(* Logix 5000 project; controller PROJECT2 Emulate 5570 rev 30.12; software revision 30.01; part 2 of 3 *)

ADD_ON_INSTRUCTION AOI_SIMAnalogSensor_OnOff   (* revision 1.0 *)
VAR_IN_OUT
   Sensor : REAL; {required}
END_VAR
VAR_INPUT
   RampUpTime : DINT; {required}
   RampDwnTime : DINT; {required}
   Min : REAL; {required}
   Max : REAL; {required}
   Target : REAL; {visible}
   Tolerance : REAL; {visible}
   Fluctuation : REAL; {access None, visible}
   Activate : BOOL; {access None}
END_VAR
VAR
   RampUpTimer : TIMER; {access None}
   RampDwnTimer : TIMER; {access None}
   FluctuateTimer : TIMER; {access None}
   FluctuateONS : BOOL; {access None}
   CurrentValue : REAL; {access Read Only}
   RampDwnTriggerONS : BOOL; {access Read Only}
   RampDwnTriggerPulse : BOOL; {access Read Only}
   RampUpTriggerONS : BOOL; {access Read Only}
   RampUpTriggerPulse : BOOL; {access Read Only}
   RandomNumber : DINT; {access Read Only}
   RandomTarget : REAL; {access Read Only}
   RandomIntermediate : DINT; {access Read Only}
   ScaledRampDwnTime : REAL; {access Read Only}
   ScaledRampUpTime : REAL; {access Read Only}
   Fluctuate : BOOL; {access None}
   LowerTargetTriggerONS : BOOL; {access None}
   OldTarget : REAL; {access None}
   RaiseTargetTriggerONS : BOOL; {access None}
END_VAR

ROUTINE Logic   (* ladder *)
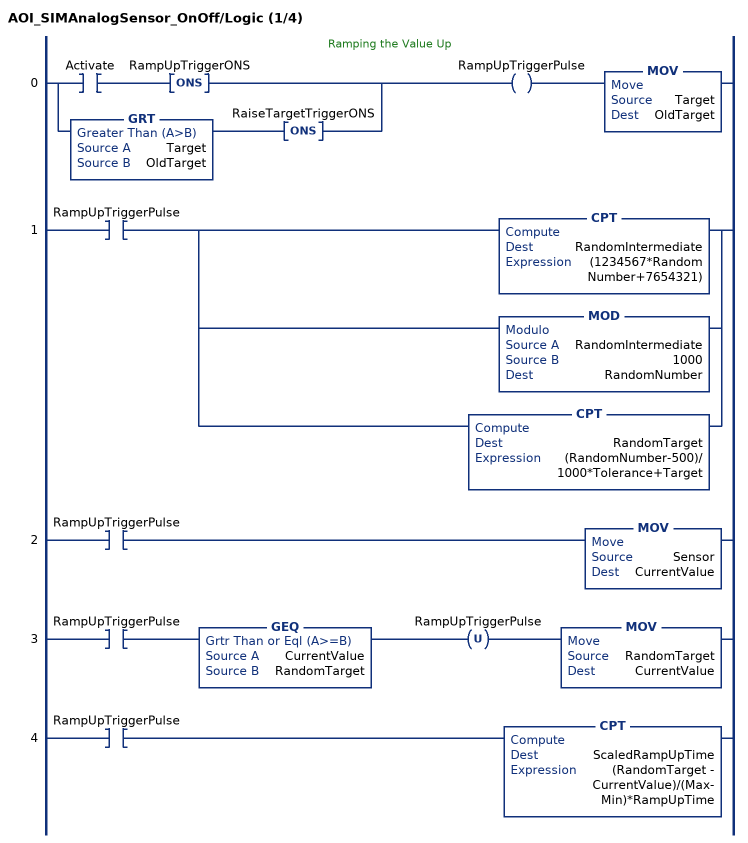
   // Ramping the Value Up
   0: [XIC(Activate) ONS(RampUpTriggerONS) ,GRT(Target,OldTarget) ONS(RaiseTargetTriggerONS) ]OTE(RampUpTriggerPulse)MOV(Target,OldTarget);
   1: XIC(RampUpTriggerPulse)[CPT(RandomIntermediate,(1234567*RandomNumber+7654321)) ,MOD(RandomIntermediate,1000,RandomNumber) ,CPT(RandomTarget,(RandomNumber-500)/1000*Tolerance+Target) ];
   2: XIC(RampUpTriggerPulse)MOV(Sensor,CurrentValue);
   3: XIC(RampUpTriggerPulse)GEQ(CurrentValue,RandomTarget)OTU(RampUpTriggerPulse)MOV(RandomTarget,CurrentValue);
   4: XIC(RampUpTriggerPulse)CPT(ScaledRampUpTime,(RandomTarget - CurrentValue)/(Max-Min)*RampUpTime);
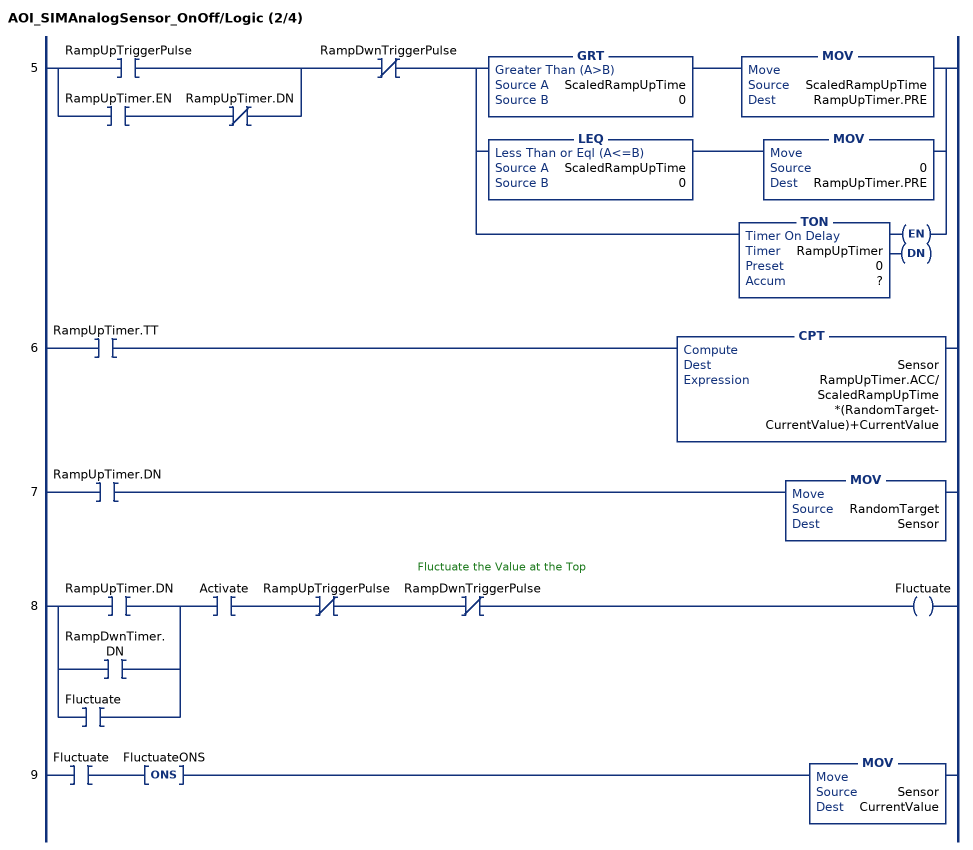
   5: [XIC(RampUpTriggerPulse) ,XIC(RampUpTimer.EN) XIO(RampUpTimer.DN) ]XIO(RampDwnTriggerPulse)[GRT(ScaledRampUpTime,0) MOV(ScaledRampUpTime,RampUpTimer.PRE) ,LEQ(ScaledRampUpTime,0) MOV(0,RampUpTimer.PRE) ,TON(RampUpTimer,?,?) ];
   6: XIC(RampUpTimer.TT)CPT(Sensor,RampUpTimer.ACC/ScaledRampUpTime *(RandomTarget-CurrentValue)+CurrentValue);
   7: XIC(RampUpTimer.DN)MOV(RandomTarget,Sensor);
   // Fluctuate the Value at the Top
   8: [XIC(RampUpTimer.DN) ,XIC(RampDwnTimer.DN) ,XIC(Fluctuate) ]XIC(Activate)XIO(RampUpTriggerPulse)XIO(RampDwnTriggerPulse)OTE(Fluctuate);
   9: XIC(Fluctuate)ONS(FluctuateONS)MOV(Sensor,CurrentValue);
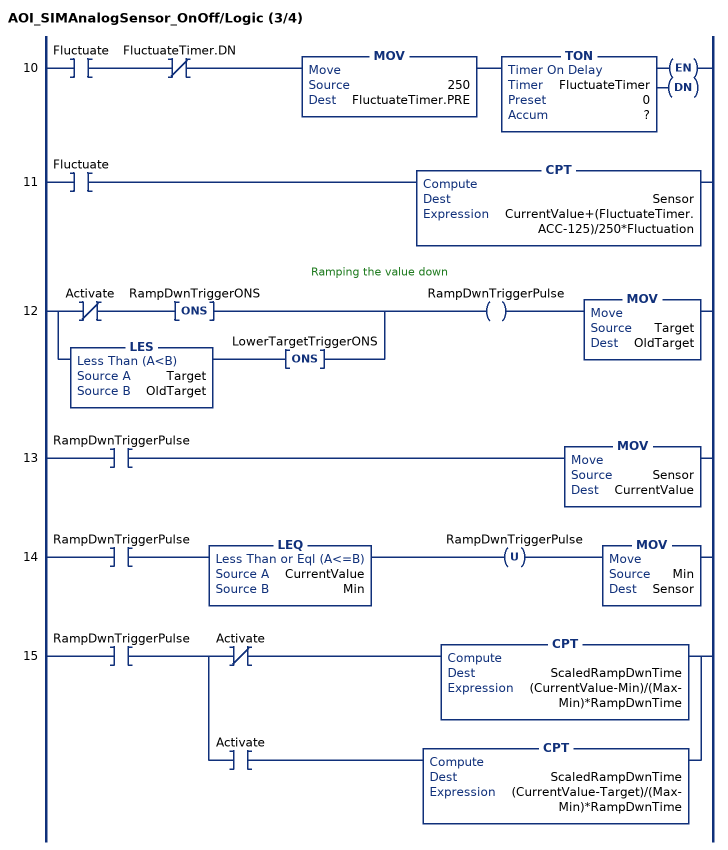
   10: XIC(Fluctuate)XIO(FluctuateTimer.DN)MOV(250,FluctuateTimer.PRE)TON(FluctuateTimer,?,?);
   11: XIC(Fluctuate)CPT(Sensor,CurrentValue+(FluctuateTimer.ACC-125)/250*Fluctuation);
   // Ramping the value down
   12: [XIO(Activate) ONS(RampDwnTriggerONS) ,LES(Target,OldTarget) ONS(LowerTargetTriggerONS) ]OTE(RampDwnTriggerPulse)MOV(Target,OldTarget);
   13: XIC(RampDwnTriggerPulse)MOV(Sensor,CurrentValue);
   14: XIC(RampDwnTriggerPulse)LEQ(CurrentValue,Min)OTU(RampDwnTriggerPulse)MOV(Min,Sensor);
   15: XIC(RampDwnTriggerPulse)[XIO(Activate) CPT(ScaledRampDwnTime,(CurrentValue-Min)/(Max-Min)*RampDwnTime) ,XIC(Activate) CPT(ScaledRampDwnTime,(CurrentValue-Target)/(Max-Min)*RampDwnTime) ];
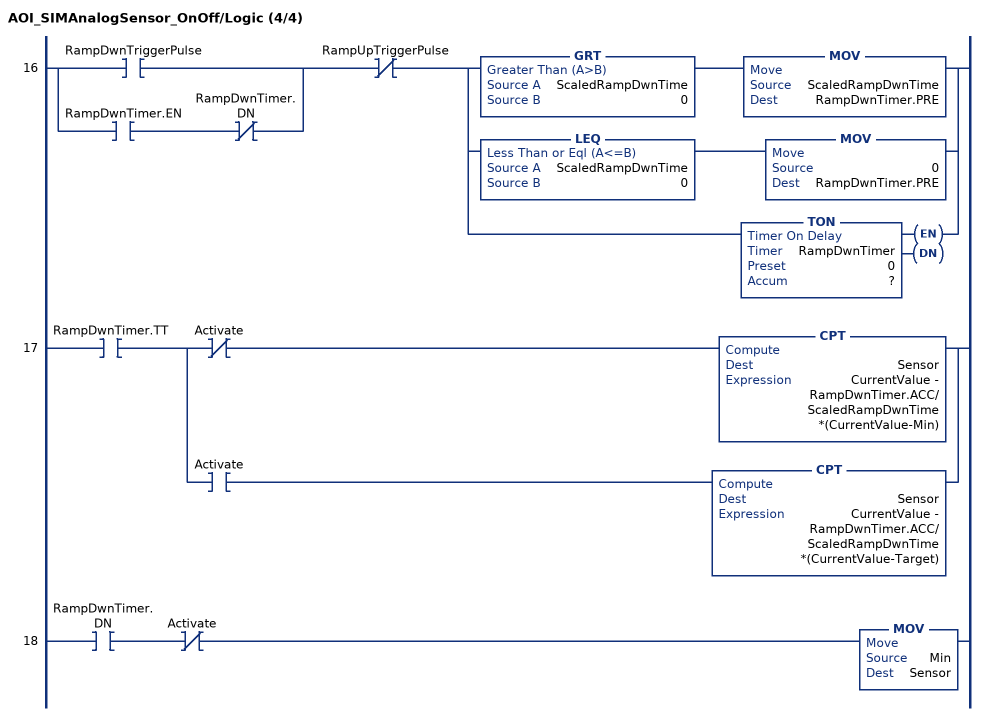
   16: [XIC(RampDwnTriggerPulse) ,XIC(RampDwnTimer.EN) XIO(RampDwnTimer.DN) ]XIO(RampUpTriggerPulse)[GRT(ScaledRampDwnTime,0) MOV(ScaledRampDwnTime,RampDwnTimer.PRE) ,LEQ(ScaledRampDwnTime,0) MOV(0,RampDwnTimer.PRE) ,TON(RampDwnTimer,?,?) ];
   17: XIC(RampDwnTimer.TT)[XIO(Activate) CPT(Sensor,CurrentValue - RampDwnTimer.ACC/ScaledRampDwnTime *(CurrentValue-Min)) ,XIC(Activate) CPT(Sensor,CurrentValue - RampDwnTimer.ACC/ScaledRampDwnTime *(CurrentValue-Target)) ];
   18: XIC(RampDwnTimer.DN)XIO(Activate)MOV(Min,Sensor);
END_ROUTINE
END_ADD_ON_INSTRUCTION

ADD_ON_INSTRUCTION AOI_SIMAnalogSensor_Profile   (* revision 1.0 *)
VAR_IN_OUT
   Sensor : REAL; {required}
END_VAR
VAR_INPUT
   RampUpTime : DINT; {required}
   RampDwnTime : DINT; {required}
   Min : REAL; {required}
   Max : REAL; {required}
   Target : REAL; {visible}
   Tolerance : REAL; {visible}
   Fluctuation : REAL; {access None, visible}
   Activate : BOOL; {access None}
END_VAR
VAR
   RampUpTimer : TIMER; {access None}
   RampDwnTimer : TIMER; {access None}
   FluctuateTimer : TIMER; {access None}
   FluctuateONS : BOOL; {access None}
   CurrentValue : REAL; {access Read Only}
   RampDwnTriggerONS : BOOL; {access Read Only}
   RampDwnTriggerPulse : BOOL; {access Read Only}
   RampUpTriggerONS : BOOL; {access Read Only}
   RampTriggerPulse : BOOL; {access Read Only}
   RandomNumber : DINT; {access Read Only}
   RandomTarget : REAL; {access Read Only}
   RandomIntermediate : DINT; {access Read Only}
   ScaledRampDwnTime : REAL; {access Read Only}
   ScaledRampUpTime : REAL; {access Read Only}
   Fluctuate : BOOL; {access None}
   LowerTargetTriggerONS : BOOL; {access None}
   OldTarget : REAL; {access None}
   RaiseTargetTriggerONS : BOOL; {access None}
END_VAR

ROUTINE Logic   (* ladder *)
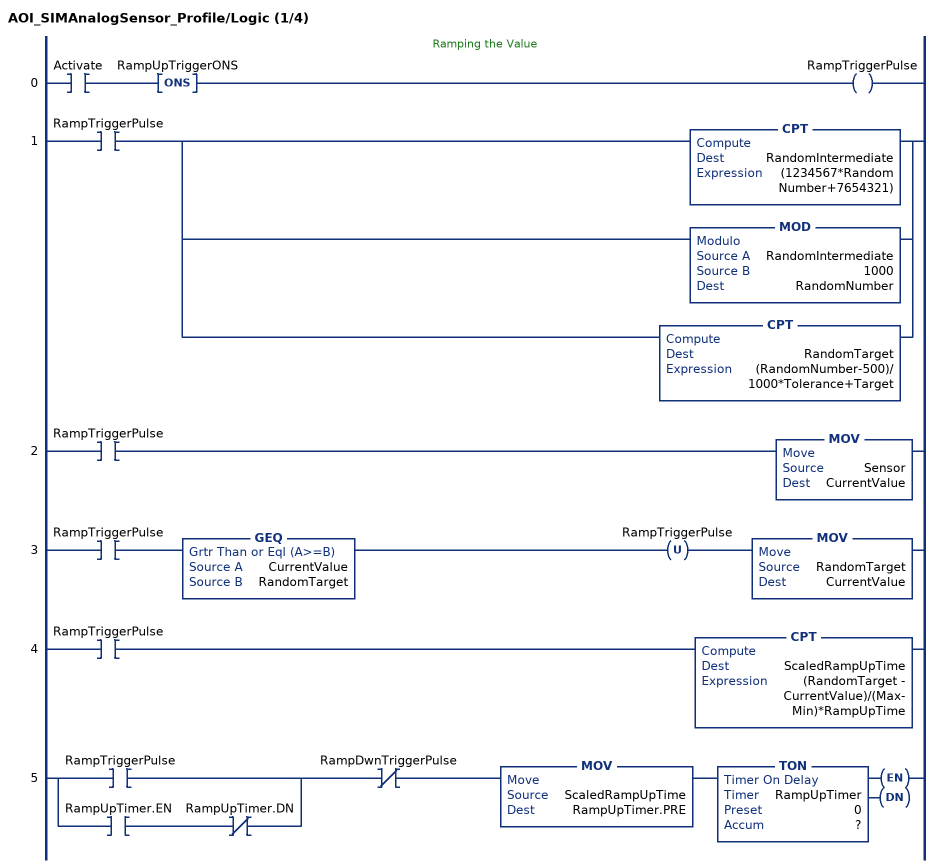
   // Ramping the Value
   0: XIC(Activate)ONS(RampUpTriggerONS)OTE(RampTriggerPulse);
   1: XIC(RampTriggerPulse)[CPT(RandomIntermediate,(1234567*RandomNumber+7654321)) ,MOD(RandomIntermediate,1000,RandomNumber) ,CPT(RandomTarget,(RandomNumber-500)/1000*Tolerance+Target) ];
   2: XIC(RampTriggerPulse)MOV(Sensor,CurrentValue);
   3: XIC(RampTriggerPulse)GEQ(CurrentValue,RandomTarget)OTU(RampTriggerPulse)MOV(RandomTarget,CurrentValue);
   4: XIC(RampTriggerPulse)CPT(ScaledRampUpTime,(RandomTarget - CurrentValue)/(Max-Min)*RampUpTime);
   5: [XIC(RampTriggerPulse) ,XIC(RampUpTimer.EN) XIO(RampUpTimer.DN) ]XIO(RampDwnTriggerPulse)MOV(ScaledRampUpTime,RampUpTimer.PRE)TON(RampUpTimer,?,?);
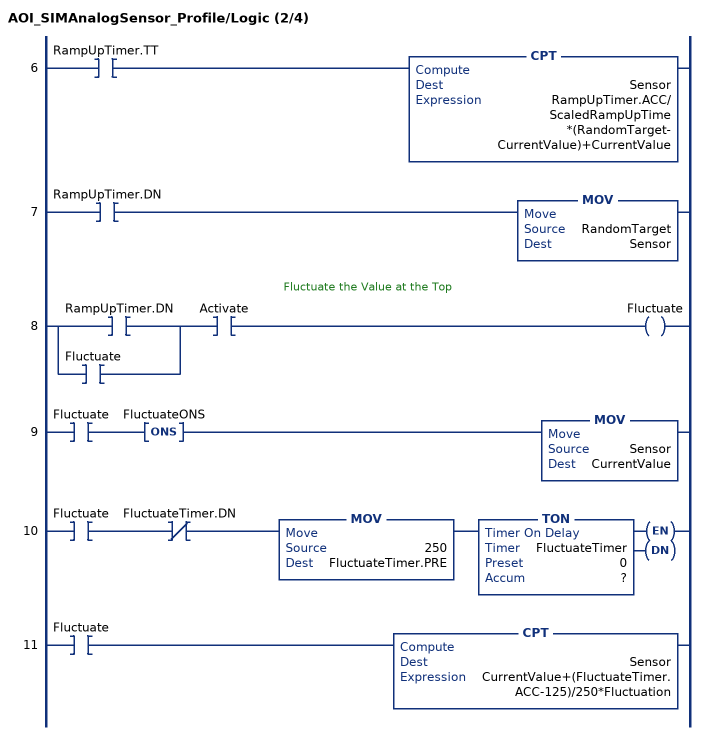
   6: XIC(RampUpTimer.TT)CPT(Sensor,RampUpTimer.ACC/ScaledRampUpTime *(RandomTarget-CurrentValue)+CurrentValue);
   7: XIC(RampUpTimer.DN)MOV(RandomTarget,Sensor);
   // Fluctuate the Value at the Top
   8: [XIC(RampUpTimer.DN) ,XIC(Fluctuate) ]XIC(Activate)OTE(Fluctuate);
   9: XIC(Fluctuate)ONS(FluctuateONS)MOV(Sensor,CurrentValue);
   10: XIC(Fluctuate)XIO(FluctuateTimer.DN)MOV(250,FluctuateTimer.PRE)TON(FluctuateTimer,?,?);
   11: XIC(Fluctuate)CPT(Sensor,CurrentValue+(FluctuateTimer.ACC-125)/250*Fluctuation);
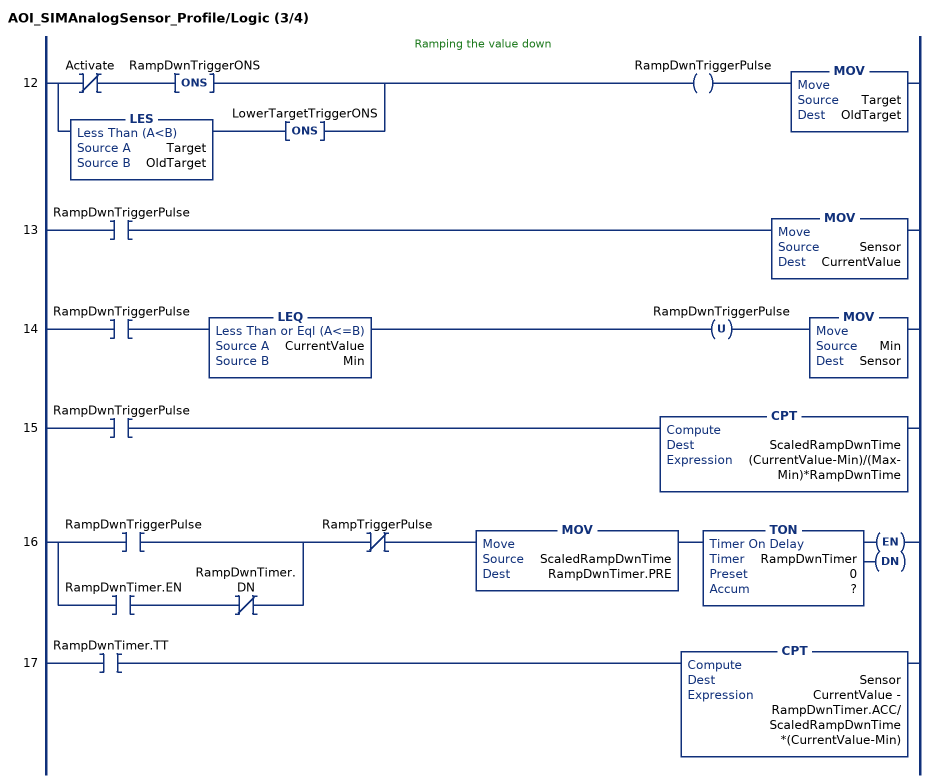
   // Ramping the value down
   12: [XIO(Activate) ONS(RampDwnTriggerONS) ,LES(Target,OldTarget) ONS(LowerTargetTriggerONS) ]OTE(RampDwnTriggerPulse)MOV(Target,OldTarget);
   13: XIC(RampDwnTriggerPulse)MOV(Sensor,CurrentValue);
   14: XIC(RampDwnTriggerPulse)LEQ(CurrentValue,Min)OTU(RampDwnTriggerPulse)MOV(Min,Sensor);
   15: XIC(RampDwnTriggerPulse)CPT(ScaledRampDwnTime,(CurrentValue-Min)/(Max-Min)*RampDwnTime);
   16: [XIC(RampDwnTriggerPulse) ,XIC(RampDwnTimer.EN) XIO(RampDwnTimer.DN) ]XIO(RampTriggerPulse)MOV(ScaledRampDwnTime,RampDwnTimer.PRE)TON(RampDwnTimer,?,?);
   17: XIC(RampDwnTimer.TT)CPT(Sensor,CurrentValue - RampDwnTimer.ACC/ScaledRampDwnTime *(CurrentValue-Min));
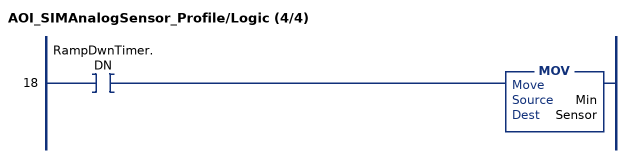
   18: XIC(RampDwnTimer.DN)MOV(Min,Sensor);
END_ROUTINE
END_ADD_ON_INSTRUCTION

ADD_ON_INSTRUCTION AOI_SIMPartSensor   (* revision 1.0 *)
VAR_OUTPUT
   Animation : DINT; {access Read Only, visible}
   Sensor : BOOL; {access Read Only, visible}
END_VAR
VAR_INPUT
   TP_ToggleSensorPB : BOOL;
   SensorON : BOOL;
   SensorOFF : BOOL;
   ONDelayTime : DINT; {visible}
   OFFDelayTime : DINT; {visible}
END_VAR
VAR_OUTPUT
   Sensor_Input : BOOL; {access Read Only, required}
END_VAR
VAR_INPUT
   SimEnabled : BOOL; {required}
   SensorONPause : BOOL;
   SensorOFFPause : BOOL;
END_VAR
VAR
   TmrON : TIMER; {access None}
   TmrOFF : TIMER; {access None}
   TP_AutoToggleSensorOFFPulse : BOOL; {access None}
   TP_AutoToggleSensorONPulse : BOOL; {access None}
   TP_AutoToggleSensorON_ONS : BOOL; {access None}
   TP_AutoToggleSensorOFF_ONS : BOOL; {access None}
   SensorOFF_ONS : BOOL; {access None}
   SensorON_ONS : BOOL; {access None}
   SensorWaitingToTurnON : BOOL; {access None}
   SensorWaitingToTurnOFF : BOOL; {access None}
   TP_ManualToggleSensorON_PULSE : BOOL; {access None}
   TP_ManualToggleSensor_ONS : BOOL; {access None}
   TP_ManualToggleSensorOFF_PULSE : BOOL; {access None}
   TP_ManualToggleSensorOFF_ONS : BOOL; {access None}
END_VAR

ROUTINE Logic   (* ladder *)
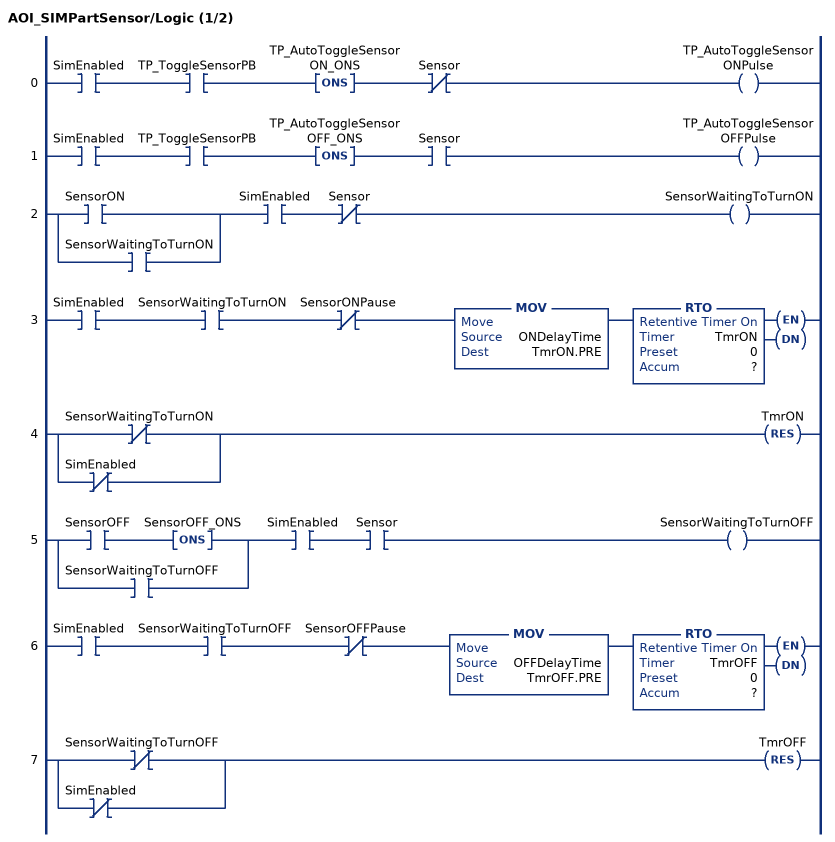
   0: XIC(SimEnabled)XIC(TP_ToggleSensorPB)ONS(TP_AutoToggleSensorON_ONS)XIO(Sensor)OTE(TP_AutoToggleSensorONPulse);
   1: XIC(SimEnabled)XIC(TP_ToggleSensorPB)ONS(TP_AutoToggleSensorOFF_ONS)XIC(Sensor)OTE(TP_AutoToggleSensorOFFPulse);
   2: [XIC(SensorON) ,XIC(SensorWaitingToTurnON) ]XIC(SimEnabled)XIO(Sensor)OTE(SensorWaitingToTurnON);
   3: XIC(SimEnabled)XIC(SensorWaitingToTurnON)XIO(SensorONPause)MOV(ONDelayTime,TmrON.PRE)RTO(TmrON,?,?);
   4: [XIO(SensorWaitingToTurnON) ,XIO(SimEnabled) ]RES(TmrON);
   5: [XIC(SensorOFF) ONS(SensorOFF_ONS) ,XIC(SensorWaitingToTurnOFF) ]XIC(SimEnabled)XIC(Sensor)OTE(SensorWaitingToTurnOFF);
   6: XIC(SimEnabled)XIC(SensorWaitingToTurnOFF)XIO(SensorOFFPause)MOV(OFFDelayTime,TmrOFF.PRE)RTO(TmrOFF,?,?);
   7: [XIO(SensorWaitingToTurnOFF) ,XIO(SimEnabled) ]RES(TmrOFF);
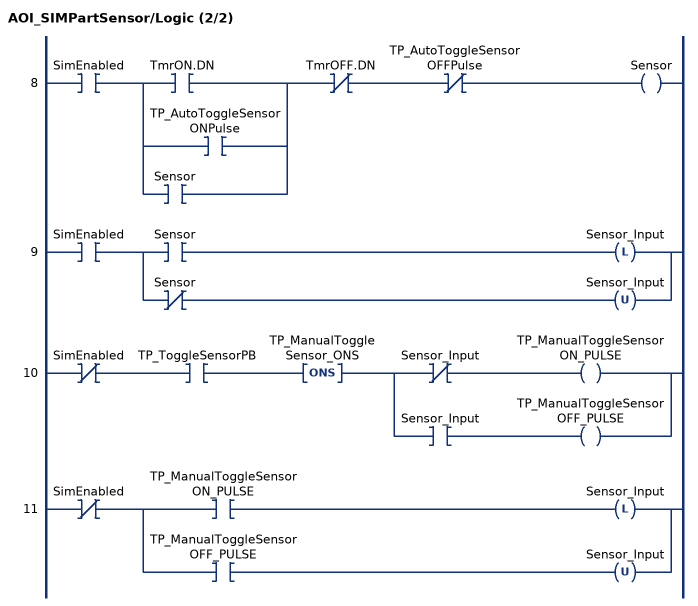
   8: XIC(SimEnabled)[XIC(TmrON.DN) ,XIC(TP_AutoToggleSensorONPulse) ,XIC(Sensor) ]XIO(TmrOFF.DN)XIO(TP_AutoToggleSensorOFFPulse)OTE(Sensor);
   9: XIC(SimEnabled)[XIC(Sensor) OTL(Sensor_Input) ,XIO(Sensor) OTU(Sensor_Input) ];
   10: XIO(SimEnabled)XIC(TP_ToggleSensorPB)ONS(TP_ManualToggleSensor_ONS)[XIO(Sensor_Input) OTE(TP_ManualToggleSensorON_PULSE) ,XIC(Sensor_Input) OTE(TP_ManualToggleSensorOFF_PULSE) ];
   11: XIO(SimEnabled)[XIC(TP_ManualToggleSensorON_PULSE) OTL(Sensor_Input) ,XIC(TP_ManualToggleSensorOFF_PULSE) OTU(Sensor_Input) ];
END_ROUTINE
END_ADD_ON_INSTRUCTION

ADD_ON_INSTRUCTION AOI_SIMPartTravel   (* revision 1.0 *)
VAR_OUTPUT
   Travelling : BOOL; {access Read Only, visible}
END_VAR
VAR_INPUT
   TravelTime : DINT; {required}
END_VAR
VAR_OUTPUT
   Animation : DINT; {access Read Only, visible}
END_VAR
VAR_INPUT
   TP_PB : BOOL;
   TravelON : BOOL;
   TravelOFF : BOOL;
   SimEnabled : BOOL; {required}
END_VAR
VAR_OUTPUT
   TravellingFirstHalf : BOOL; {access Read Only}
   TravellingLastHalf : BOOL; {access Read Only}
   TravellingLastQuarter : BOOL; {access Read Only}
   TravellingFirstQuarter : BOOL; {access Read Only}
   TravellingFirst10Percent : BOOL; {access Read Only}
   TravellingLast10Percent : BOOL; {access Read Only}
END_VAR
VAR_INPUT
   Pause : BOOL;
END_VAR
VAR_OUTPUT
   Done : BOOL; {access Read Only}
END_VAR
VAR
   Tmr : TIMER := (PRE := 1500); {access None}
   TravelON_ONS : BOOL; {access None}
   TravelTime75Percent : DINT; {access None}
   TravelTime50Percent : DINT; {access None}
   TravelTime25Percent : DINT; {access None}
   TravelTime10Percent : DINT; {access Read Only}
   TravelTime90Percent : DINT; {access Read Only}
   DonePulse : TIMER := (PRE := 250); {access None}
   TP_AutoToggleTravellingON_ONS : BOOL; {access None}
   TP_AutoToggleTravellingONPulse : BOOL; {access None}
   TP_AutoToggleTravellingOFFPulse : BOOL; {access None}
   TP_AutoToggleTravellingOFF_ONS : BOOL; {access None}
END_VAR

ROUTINE Logic   (* ladder *)
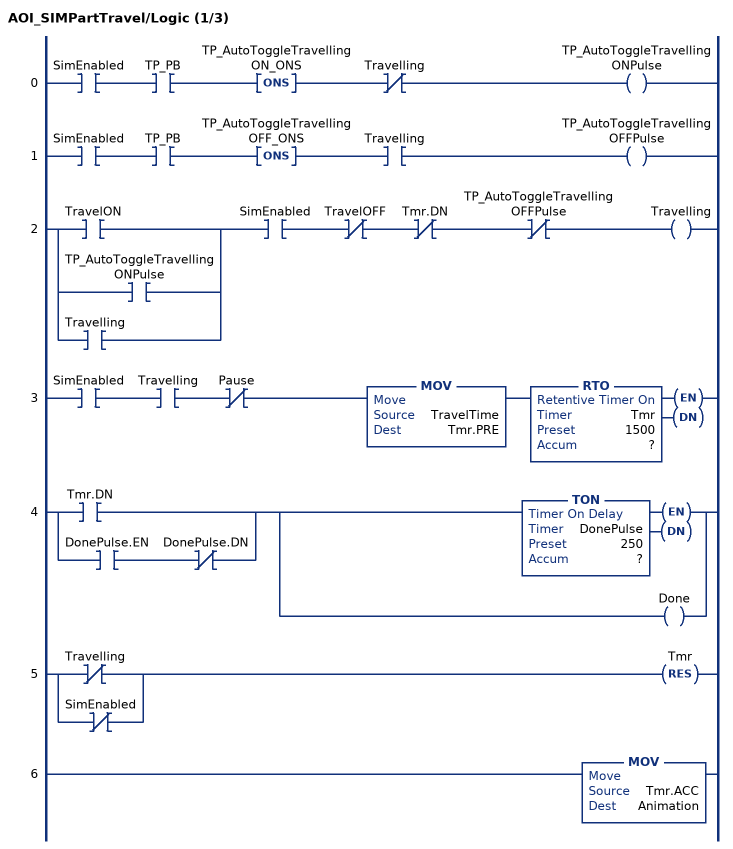
   0: XIC(SimEnabled)XIC(TP_PB)ONS(TP_AutoToggleTravellingON_ONS)XIO(Travelling)OTE(TP_AutoToggleTravellingONPulse);
   1: XIC(SimEnabled)XIC(TP_PB)ONS(TP_AutoToggleTravellingOFF_ONS)XIC(Travelling)OTE(TP_AutoToggleTravellingOFFPulse);
   2: [XIC(TravelON) ,XIC(TP_AutoToggleTravellingONPulse) ,XIC(Travelling) ]XIC(SimEnabled)XIO(TravelOFF)XIO(Tmr.DN)XIO(TP_AutoToggleTravellingOFFPulse)OTE(Travelling);
   3: XIC(SimEnabled)XIC(Travelling)XIO(Pause)MOV(TravelTime,Tmr.PRE)RTO(Tmr,?,?);
   4: [XIC(Tmr.DN) ,XIC(DonePulse.EN) XIO(DonePulse.DN) ][TON(DonePulse,?,?) ,OTE(Done) ];
   5: [XIO(Travelling) ,XIO(SimEnabled) ]RES(Tmr);
   6: MOV(Tmr.ACC,Animation);
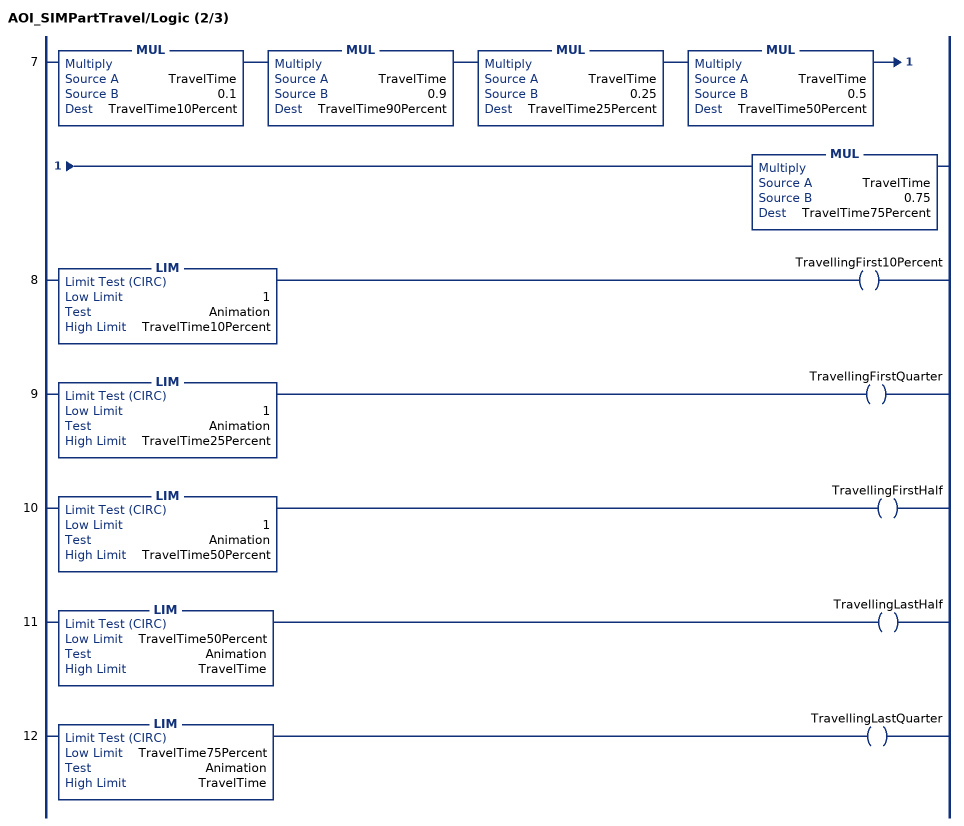
   7: MUL(TravelTime,0.1,TravelTime10Percent)MUL(TravelTime,0.9,TravelTime90Percent)MUL(TravelTime,0.25,TravelTime25Percent)MUL(TravelTime,0.5,TravelTime50Percent)MUL(TravelTime,0.75,TravelTime75Percent);
   8: LIM(1,Animation,TravelTime10Percent)OTE(TravellingFirst10Percent);
   9: LIM(1,Animation,TravelTime25Percent)OTE(TravellingFirstQuarter);
   10: LIM(1,Animation,TravelTime50Percent)OTE(TravellingFirstHalf);
   11: LIM(TravelTime50Percent,Animation,TravelTime)OTE(TravellingLastHalf);
   12: LIM(TravelTime75Percent,Animation,TravelTime)OTE(TravellingLastQuarter);
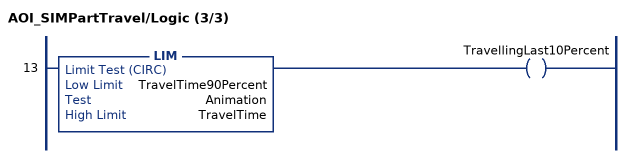
   13: LIM(TravelTime90Percent,Animation,TravelTime)OTE(TravellingLast10Percent);
END_ROUTINE
END_ADD_ON_INSTRUCTION

VAR_GLOBAL   (* controller tags *)
   AVG_CYCLE_TIME : DINT;
   CAP_FAULT_ONESHOT5 : BOOL;
   CAPFAULTTIMER : TIMER := (PRE := 4000);
   CAPINSERTTIMER : TIMER := (PRE := 500);
   CapSecured : ALIAS FOR TP.PLC.YELLOW.LT;
   CH0 : ALIAS FOR Local:4:I.Ch0Data;
   CH1 : ALIAS FOR Local:4:I.Ch1Data;
   CURRENT_CYCLE_TIME : DINT;
   CURRENT_NO_BOTTLES : DINT;
   FILL_COMPLE_TIMER : TIMER := (PRE := 2000);
   FILL_LEVEL : REAL;
   FillComplete : ALIAS FOR TP.PLC.BLUE.LT;
   FILLSENSDELAYTIMER : TIMER := (PRE := 500);
   I2 : ALIAS FOR Local:2:I.Data;
        .0   // START BUTTON
        .5   // POWER ON BUTTON
        .1   // STOP BUTTON
   I31 : ALIAS FOR Ethernet3_PointIO:1:I;
        .6   // BOTTLE AT POSITON 1
        .2   // EXTENDED POSITION
        .3   // RETRACTED POSITION
        .0   // clamped position
        .1   // UNCLAMP
   I32 : ALIAS FOR Ethernet3_PointIO:2:I;
        .2   // FILL SENSOR
        .5   // CAP CHECK
        .7   // BOTTLE AT STATION 3
        .1   // SOLINOID AT RAISED POSTION
        .6   // CAP LOWER POSITION
   I33 : ALIAS FOR Ethernet3_PointIO:3:I;
        .1   // UPPER POSITION
        .6   // BOTTLE AT POSITION 5
        .0   // SOLINOID LOWER POSITION
        .2   // Cap Rotating
        .3   // BOTTLE AT STATION 4
   MAX_LEVEL : REAL;
   MAXLEVL_ONESHOT1 : BOOL;
   MAXLVL_ONESHOT1 : BOOL;
   NO_OF_BOTTLES : COUNTER := (PRE := 999999999);
   NOOFBOT_ONESHOT3 : BOOL;
   O3 : ALIAS FOR Local:3:O.Data;
        .0   // START LIGHT
   O34 : ALIAS FOR Ethernet3_PointIO:4:O;
        .1   // UNCLAMP
        .0   // CLAMP
        .2   // EXTEND WALKING BEAM
        .3   // RETRACTION
   O35 : ALIAS FOR Ethernet3_PointIO:5:O;
        .0   // LOWER SOLINOID
        .1   // FILL BOTTLE
        .6   // CAP INSERT LOWER
   O36 : ALIAS FOR Ethernet3_PointIO:6:O;
        .0   // CAP INSERT LOWER
        .1   // CAP INSERT RISE
        .2   // ROTATION
   ONE1 : BOOL;
   ONE2 : BOOL;
   ONE3 : BOOL;
   ONE4 : BOOL;
   SPEED_SENSOR : REAL;
   TIMER : TIMER;
   TOTAL_CYCLE_TIME : DINT;
   TOTAL_CYCLE_TIMER : TIMER := (PRE := 99999999);
   TOTAL_NO_FAULTS : DINT;
   TOTAL_NO_OF_BOT : DINT;
   TOTCYCLTIME_ONESHOT2 : BOOL;
   TP : TouchPanel := (PLC.INT1_TXT := 'CURRENT CYCLE TIME IN SECONDS :', PLC.INT2_TXT := 'CURRENT NO OF BOTTLES :', PLC.INT3_TXT := 'TOTAL NO OF BOTTLES :', PLC.INT4_TXT := 'TOTAL NO FAULTS (CAP INSERTION) :', PLC.REAL1_TXT := 'FILL LEVEL SENSOR (4-20V) :', PLC.REAL2_TXT := 'SPEED SENSOR (0-10V) :', PLC.REAL3_TXT := 'MAX FILL VALUE :', PLC.REAL4_TXT := 'NOT IN USE', PLC.GRAY.PB_TXT := 'TP.PLC.GRAY.PB', PLC.GRAY.LT_TXT := 'TP.PLC.GRAY.LT', PLC.BLUE.PB_TXT := 'TP.PLC.BLUE.PB', PLC.BLUE.LT_TXT := 'TP.PLC.BLUE.LT', PLC.GREEN.PB_TXT := 'TP.PLC.GREEN.PB', PLC.GREEN.LT_TXT := 'TP.PLC.GREEN.LT', PLC.YELLOW.PB_TXT := 'TP.PLC.YELLOW.PB', PLC.YELLOW.LT_TXT := 'TP.PLC.YELLOW.LT', PLC.RED.PB_TXT := 'TP.PLC.RED.PB', PLC.RED.LT_TXT := 'TP.PLC.RED.LT', Stn.Auto.LT := 1, Stn.CycleStart.LT := 1, Stn.Lift.Lower.LT := 1, Stn.Reject.Ret.LT := 1, Stn.Divert.Ret.LT := 1, Stn.SendToConv.LT := 1, Conv.TargetSpeed := 8.0, Conv.RemCntl.On.LT := 1, Servo.Power.On.LT := 1, Servo.Feedback.On.LT := 1, Servo.Vertical.Raise.LT := 1, Servo.CurrentPostionIND := 50.0211, Servo.JogSpeed := 10.0, Servo.TargetPosition := 222.0, Servo.TargetSpeed := 50.0);
        .PLC.GREEN.LT   // GREEN TP LIGHT
END_VAR

PROGRAM MainProgram   (* main routine MainRoutine *)
VAR
   _temp : BOOL;
   SIM_BNOP : BOOL := 1;
   SIM_LevelSensor : AOI_SIMAnalogSensor_OnOff := (RampUpTime := 500, RampDwnTime := 500, Min := 4.0, Max := 20.0, Target := 17.71, Tolerance := 0.5, Fluctuation := 0.1);
   SIM_NOP : BOOL := 1;
   SIM_ONS : BOOL;
   SIM_OutfeedSensor : AOI_SIMPartSensor := (SimEnabled := 1);
   SIM_PowerONPB : BOOL;
   SIM_PPENABLED : BOOL := 1;
   SIM_PTInfeedToStn1 : AOI_SIMPartTravel := (TravelTime := 3928, SimEnabled := 1);
   SIM_PTStn2Fill : AOI_SIMPartTravel := (TravelTime := 3000, SimEnabled := 1, Pause := 1);
   SIM_PTStn4ToOutfeed : AOI_SIMPartTravel := (TravelTime := 5000, SimEnabled := 1);
   SIM_PTStnStatus : StationStatus[20] := ([1].BottlePresent := 1, [2].BottlePresent := 1, [3].BottlePresent := 1, [3].BottleFilled := 1, [4].BottlePresent := 1, [4].BottleFilled := 1, [4].CapInserted := 1, [5].BottleFilled := 1, [5].CapSecured := 1, [11].BottlePresent := 1, [12].BottlePresent := 1, [12].BottleFilled := 1, [13].BottlePresent := 1, [13].BottleFilled := 1, [13].CapInserted := 1, [14].BottlePresent := 1, [14].BottleFilled := 1, [14].CapSecured := 1, [15].BottleFilled := 1, [15].CapSecured := 1);
   SIM_PTWalkingBeam : AOI_SIMPartTravel := (TravelTime := 5000, SimEnabled := 1, Pause := 1);
   SIM_SpeedSensor : AOI_SIMAnalogSensor_OnOff := (RampUpTime := 50, RampDwnTime := 4000, Max := 10.0, Target := 8.0, Tolerance := 0.5, Fluctuation := 0.1);
   SIM_Stn1BottlePresentSensor : AOI_SIMPartSensor := (Sensor := 1, ONDelayTime := 750, OFFDelayTime := 1000, Sensor_Input := 1, SimEnabled := 1, SensorOFFPause := 1);
   SIM_Stn2BottleFilledSensor : AOI_SIMPartSensor := (SensorOFF := 1, ONDelayTime := 50, OFFDelayTime := 50, SimEnabled := 1);
   SIM_Stn2BottlePresentSensor : AOI_SIMPartSensor := (Sensor := 1, ONDelayTime := 750, OFFDelayTime := 1500, Sensor_Input := 1, SimEnabled := 1, SensorONPause := 1, SensorOFFPause := 1);
   SIM_Stn2Filler_Cylinder : AOI_SIM_2PosCyl_RsLwr := (TravelTime := 1000, Raise_Output := 1, Raise_Sensor := 1, SingleSolenoidLower := 1, Raise_Activated := 1);
   SIM_Stn2Filler_Fill : AOI_SIM_SimpleValve := (TravelTime := 1, Animation := -19);
   SIM_Stn3BottlePresentSensor : AOI_SIMPartSensor := (Sensor := 1, ONDelayTime := 1500, OFFDelayTime := 2000, Sensor_Input := 1, SimEnabled := 1, SensorONPause := 1, SensorOFFPause := 1);
   SIM_Stn3CapInsert : AOI_SIM_2PosCyl_RsLwr := (TravelTime := 1000, Animation := -15, Raise_Output := 1, Raise_Sensor := 1, SingleSolenoidLower := 1, Raise_Activated := 1);
   SIM_Stn3CapPresentSensor : AOI_SIMPartSensor := (Sensor := 1, SensorON := 1, ONDelayTime := 1500, OFFDelayTime := 50, Sensor_Input := 1, SimEnabled := 1);
   SIM_Stn4BottlePresentSensor : AOI_SIMPartSensor := (Sensor := 1, ONDelayTime := 1500, OFFDelayTime := 2000, Sensor_Input := 1, SimEnabled := 1, SensorONPause := 1, SensorOFFPause := 1);
   SIM_Stn4CapRotate : AOI_SIM_Conveyor := (RunDelay := 50);
   SIM_Stn4CapRotate_Cylinder : AOI_SIM_2PosCyl_RsLwr := (TravelTime := 3000, Raise_Sensor := 1);
   SIM_WalkingBeam : AOI_SIM_3PosCyl_ExtRet := (TravelTime := 5000, Animation := 5019, Extend_Sensor := 1);
   SIM_WalkingBeamClamp : AOI_SIM_2PosCyl_ExtRet := (TravelTime := 1000, Retract_Sensor := 1);
   SIM_Zero : DINT;
END_VAR

ROUTINE MainRoutine   (* ladder *)
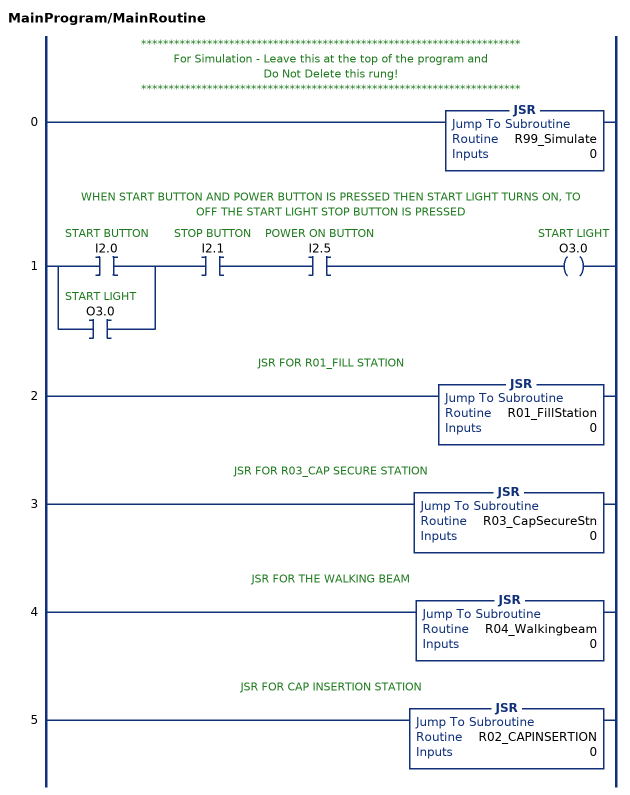
   // *********************************************************************
   // For Simulation - Leave this at the top of the program and
   // Do Not Delete this rung!
   // *********************************************************************
   0: JSR(R99_Simulate,0);
   // WHEN START BUTTON AND POWER BUTTON IS PRESSED THEN START LIGHT TURNS ON, TO OFF THE START LIGHT STOP BUTTON IS PRESSED
   1: [XIC(I2.0) ,XIC(O3.0) ]XIC(I2.1)XIC(I2.5)OTE(O3.0);
   // JSR FOR R01_FILL STATION
   2: JSR(R01_FillStation,0);
   // JSR FOR R03_CAP SECURE STATION
   3: JSR(R03_CapSecureStn,0);
   // JSR FOR THE WALKING BEAM
   4: JSR(R04_Walkingbeam,0);
   // JSR FOR CAP INSERTION STATION
   5: JSR(R02_CAPINSERTION,0);
END_ROUTINE

ROUTINE R01_FillStation   (* ladder *)
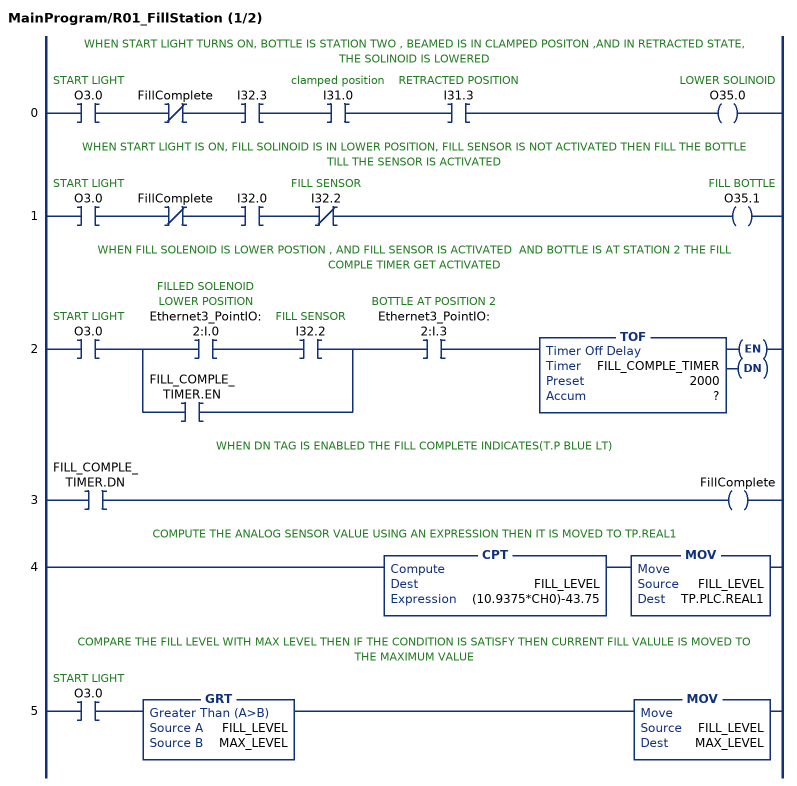
   // WHEN START LIGHT TURNS ON, BOTTLE IS STATION TWO , BEAMED IS IN CLAMPED POSITON ,AND IN RETRACTED STATE, THE SOLINOID IS LOWERED
   0: XIC(O3.0)XIO(FillComplete)XIC(I32.3)XIC(I31.0)XIC(I31.3)OTE(O35.0);
   // WHEN START LIGHT IS ON, FILL SOLINOID IS IN LOWER POSITION, FILL SENSOR IS NOT ACTIVATED THEN FILL THE BOTTLE TILL THE SENSOR IS ACTIVATED
   1: XIC(O3.0)XIO(FillComplete)XIC(I32.0)XIO(I32.2)OTE(O35.1);
   // WHEN FILL SOLENOID IS LOWER POSTION , AND FILL SENSOR IS ACTIVATED  AND BOTTLE IS AT STATION 2 THE FILL COMPLE TIMER GET ACTIVATED
   2: XIC(O3.0)[XIC(Ethernet3_PointIO:2:I.0) XIC(I32.2) ,XIC(FILL_COMPLE_TIMER.EN) ]XIC(Ethernet3_PointIO:2:I.3)TOF(FILL_COMPLE_TIMER,?,?);
   // WHEN DN TAG IS ENABLED THE FILL COMPLETE INDICATES(T.P BLUE LT)
   3: XIC(FILL_COMPLE_TIMER.DN)OTE(FillComplete);
   // COMPUTE THE ANALOG SENSOR VALUE USING AN EXPRESSION THEN IT IS MOVED TO TP.REAL1
   4: CPT(FILL_LEVEL,(10.9375*CH0)-43.75)MOV(FILL_LEVEL,TP.PLC.REAL1);
   // COMPARE THE FILL LEVEL WITH MAX LEVEL THEN IF THE CONDITION IS SATISFY THEN CURRENT FILL VALULE IS MOVED TO THE MAXIMUM VALUE
   5: XIC(O3.0)GRT(FILL_LEVEL,MAX_LEVEL)MOV(FILL_LEVEL,MAX_LEVEL);
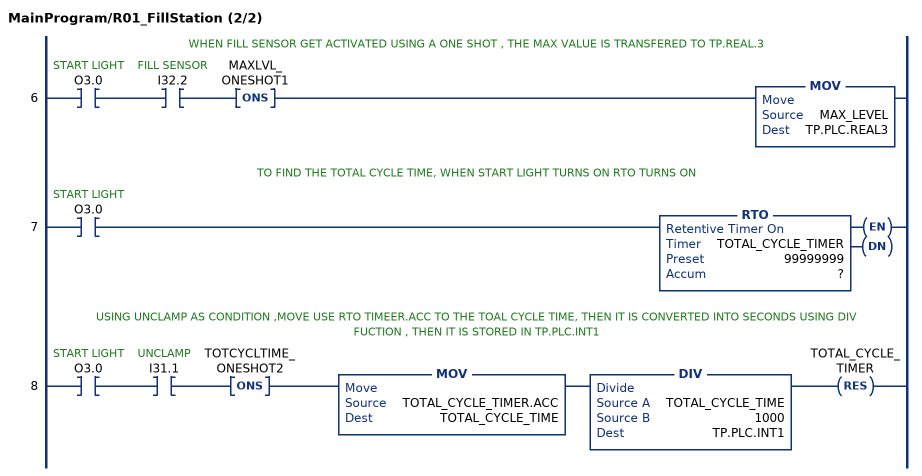
   // WHEN FILL SENSOR GET ACTIVATED USING A ONE SHOT , THE MAX VALUE IS TRANSFERED TO TP.REAL.3
   6: XIC(O3.0)XIC(I32.2)ONS(MAXLVL_ONESHOT1)MOV(MAX_LEVEL,TP.PLC.REAL3);
   // TO FIND THE TOTAL CYCLE TIME, WHEN START LIGHT TURNS ON RTO TURNS ON
   7: XIC(O3.0)RTO(TOTAL_CYCLE_TIMER,?,?);
   // USING UNCLAMP AS CONDITION ,MOVE USE RTO TIMEER.ACC TO THE TOAL CYCLE TIME, THEN IT IS CONVERTED INTO SECONDS USING DIV FUCTION , THEN IT IS STORED IN TP.PLC.INT1
   8: XIC(O3.0)XIC(I31.1)ONS(TOTCYCLTIME_ONESHOT2)MOV(TOTAL_CYCLE_TIMER.ACC,TOTAL_CYCLE_TIME)DIV(TOTAL_CYCLE_TIME,1000,TP.PLC.INT1)RES(TOTAL_CYCLE_TIMER);
END_ROUTINE

ROUTINE R02_CAPINSERTION   (* ladder *)
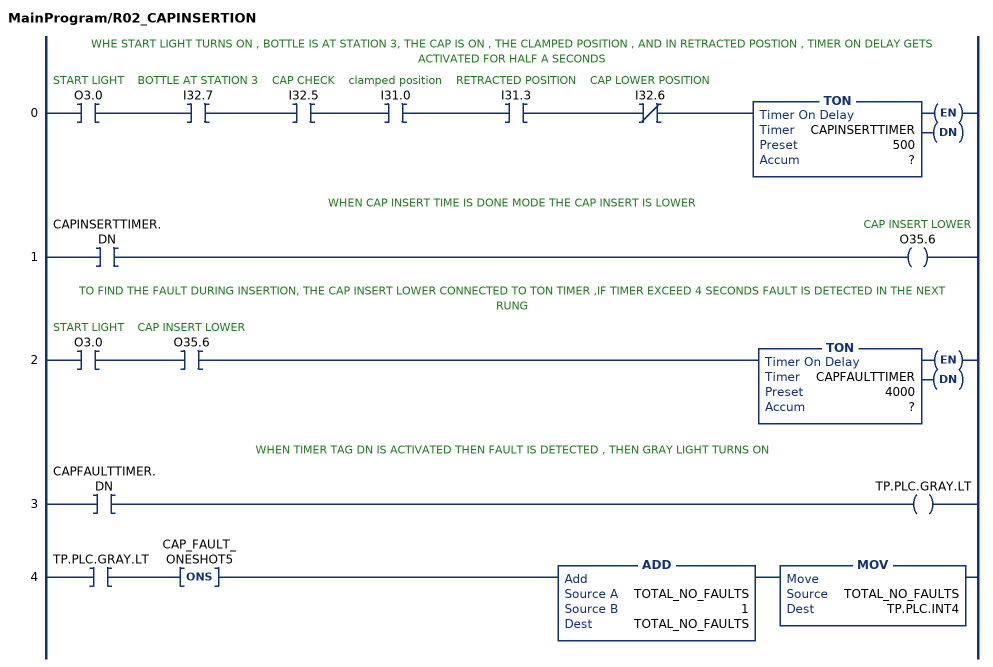
   // WHE START LIGHT TURNS ON , BOTTLE IS AT STATION 3, THE CAP IS ON , THE CLAMPED POSITION , AND IN RETRACTED POSTION , TIMER ON DELAY GETS ACTIVATED FOR HALF A SECONDS
   0: XIC(O3.0)XIC(I32.7)XIC(I32.5)XIC(I31.0)XIC(I31.3)XIO(I32.6)TON(CAPINSERTTIMER,?,?);
   // WHEN CAP INSERT TIME IS DONE MODE THE CAP INSERT IS LOWER
   1: XIC(CAPINSERTTIMER.DN)OTE(O35.6);
   // TO FIND THE FAULT DURING INSERTION, THE CAP INSERT LOWER CONNECTED TO TON TIMER ,IF TIMER EXCEED 4 SECONDS FAULT IS DETECTED IN THE NEXT RUNG
   2: XIC(O3.0)XIC(O35.6)TON(CAPFAULTTIMER,?,?);
   // WHEN TIMER TAG DN IS ACTIVATED THEN FAULT IS DETECTED , THEN GRAY LIGHT TURNS ON
   3: XIC(CAPFAULTTIMER.DN)OTE(TP.PLC.GRAY.LT);
   4: XIC(TP.PLC.GRAY.LT)ONS(CAP_FAULT_ONESHOT5)ADD(TOTAL_NO_FAULTS,1,TOTAL_NO_FAULTS)MOV(TOTAL_NO_FAULTS,TP.PLC.INT4);
END_ROUTINE

ROUTINE R03_CapSecureStn   (* ladder *)
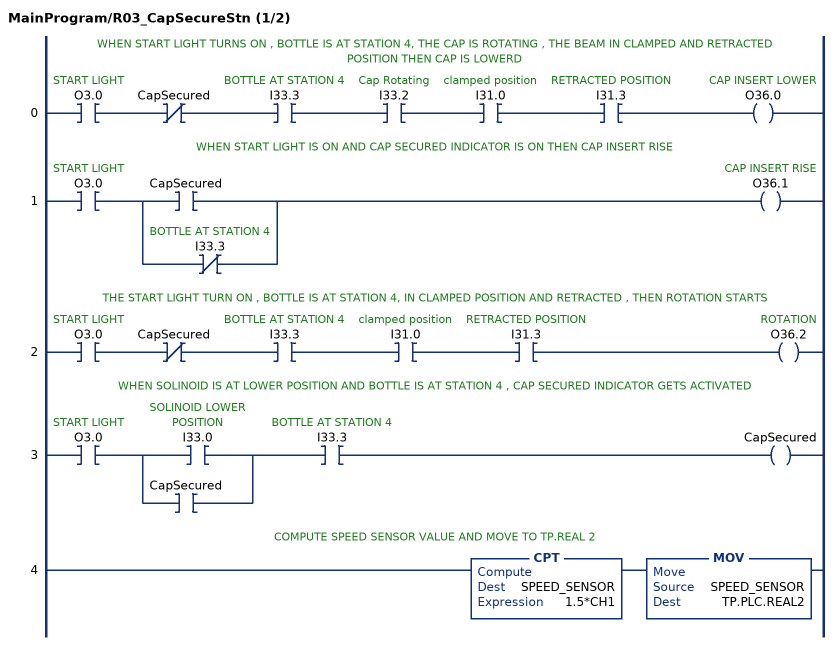
   // WHEN START LIGHT TURNS ON , BOTTLE IS AT STATION 4, THE CAP IS ROTATING , THE BEAM IN CLAMPED AND RETRACTED POSITION THEN CAP IS LOWERD
   0: XIC(O3.0)XIO(CapSecured)XIC(I33.3)XIC(I33.2)XIC(I31.0)XIC(I31.3)OTE(O36.0);
   // WHEN START LIGHT IS ON AND CAP SECURED INDICATOR IS ON THEN CAP INSERT RISE
   1: XIC(O3.0)[XIC(CapSecured) ,XIO(I33.3) ]OTE(O36.1);
   // THE START LIGHT TURN ON , BOTTLE IS AT STATION 4, IN CLAMPED POSITION AND RETRACTED , THEN ROTATION STARTS
   2: XIC(O3.0)XIO(CapSecured)XIC(I33.3)XIC(I31.0)XIC(I31.3)OTE(O36.2);
   // WHEN SOLINOID IS AT LOWER POSITION AND BOTTLE IS AT STATION 4 , CAP SECURED INDICATOR GETS ACTIVATED
   3: XIC(O3.0)[XIC(I33.0) ,XIC(CapSecured) ]XIC(I33.3)OTE(CapSecured);
   // COMPUTE SPEED SENSOR VALUE AND MOVE TO TP.REAL 2
   4: CPT(SPEED_SENSOR,1.5*CH1)MOV(SPEED_SENSOR,TP.PLC.REAL2);
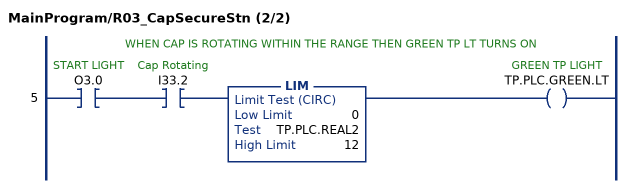
   // WHEN CAP IS ROTATING WITHIN THE RANGE THEN GREEN TP LT TURNS ON
   5: XIC(O3.0)XIC(I33.2)LIM(0,TP.PLC.REAL2,12)OTE(TP.PLC.GREEN.LT);
END_ROUTINE
